FUNCTION_BLOCK FB_AppelEtage

VAR_INPUT
	bBouton : BOOL;
    iEtage  : INT;
END_VAR

VAR_OUTPUT
	bDemande : BOOL;
    iEtageDemande : INT;
END_VAR

VAR
	rTrig : R_TRIG;
END_VAR

// Détection front
rTrig(CLK := bBouton);

IF rTrig.Q THEN
    bDemande := TRUE;
    iEtageDemande := iEtage;
ELSE
    bDemande := FALSE;
END_IF;

END_FUNCTION_BLOCK

(* stored: Version 1.1.0.1, ProductVersion 3.1.4024.16
   POU FB_AppelEtage: Id {5623fef1-f5ac-4bc7-a33a-1a92002ecfee}, SpecialFunc None *)
